(* PLC project coking-refinery, Generated TextualNotationConverter 1.0 *)
(* stored: creationDateTime 2025-07-30T12:00:00, modificationDateTime 2025-01-30T12:00:00 *)

FUNCTION_BLOCK ANALOG_IN
  VAR_INPUT
    Name : STRING;
    Description : STRING;
    Raw_Signal : REAL;
    PV_High : REAL;
    PV_Low : REAL;
    Scaling_Slope : REAL;
    Scaling_Offset : REAL;
    Alarm_Enable : BOOL;
  END_VAR
  VAR_OUTPUT
    PV : REAL;
    High_Alarm : BOOL;
    Low_Alarm : BOOL;
    General_Fault : BOOL;
  END_VAR

            
          
END_FUNCTION_BLOCK

FUNCTION_BLOCK PID_BASIC
  VAR_INPUT
    Name : STRING;
    Description : STRING;
    AUTO : BOOL;
    PV : REAL;
    SP : REAL;
    MV_MIN : REAL;
    MV_MAX : REAL;
    X0 : REAL;
    KP : REAL;
    TR : REAL;
    TD : REAL;
    PV_High : REAL;
    PV_Low : REAL;
    Deviation_Limit : REAL;
    Inhibit : BOOL;
  END_VAR
  VAR_OUTPUT
    PV_High_Alarm : BOOL;
    PV_Low_Alarm : BOOL;
    Deviation_Alarm : BOOL;
    XOUT : REAL;
  END_VAR

            
          
END_FUNCTION_BLOCK

FUNCTION_BLOCK RATIO_CONTROL
  VAR_INPUT
    Name : STRING;
    Description : STRING;
    Auto : BOOL;
    PrimaryPV : REAL;
    SecondaryPV : REAL;
    RatioSP : REAL;
    Bias : REAL;
    TrimKp : REAL;
    TrimTi : STRING;
    MV_MIN : REAL;
    MV_MAX : REAL;
    ManOut : REAL;
    Inhibit : BOOL;
  END_VAR
  VAR_OUTPUT
    SlaveSP : REAL;
    ActiveRatio : REAL;
    RatioErr : REAL;
  END_VAR

            
          
END_FUNCTION_BLOCK

FUNCTION_BLOCK VALVE_ELECTRIC
  VAR_INPUT
    Name : STRING;
    Description : STRING;
    Control_Signal : REAL;
    Manual_Mode : BOOL;
    Manual_Position : REAL;
    Open_Limit : REAL;
    Close_Limit : REAL;
    Timeout : STRING;
    Inhibit : BOOL;
  END_VAR
  VAR_OUTPUT
    Valve_Position : REAL;
    Feedback_Pos : REAL;
    Valve_Moving : BOOL;
    Position_Error : BOOL;
    Alarm : BOOL;
  END_VAR

            
          
END_FUNCTION_BLOCK

PROGRAM Section2
  VAR
    FT101_FeedFlow_PV_kgphr : REAL;
    FT102_RefluxFlow_PV_kgphr : REAL;
    FFIC103_RefluxFlow_SP_kgphr : REAL;
    FIC104_Output_Percent : REAL;
    FV104_ValvePosition_Percent : REAL;
    FV104_FeedbackPos_Percent : REAL;
    FV104_ValveMoving : BOOL;
    PIT106_ColumnPressure_bar : REAL;
    TIT104_Temperature_C : REAL;
    TIT105_Temperature_C : REAL;
    TIT107_Temperature_C : REAL;
  END_VAR
  VAR
    FT-101 : ANALOG_IN;
    FT-102 : ANALOG_IN;
    PIT-106 : ANALOG_IN;
    TIT-104 : ANALOG_IN;
    TIT-105 : ANALOG_IN;
    TIT-107 : ANALOG_IN;
    FFIC-103 : RATIO_CONTROL;
    FIC-104 : PID_BASIC;
    FV-104 : VALVE_ELECTRIC;
  END_VAR
  VAR  (* added by the conversion: wires and edge detectors of the diagram *)
    _OR1_OUT : BOOL;
  END_VAR

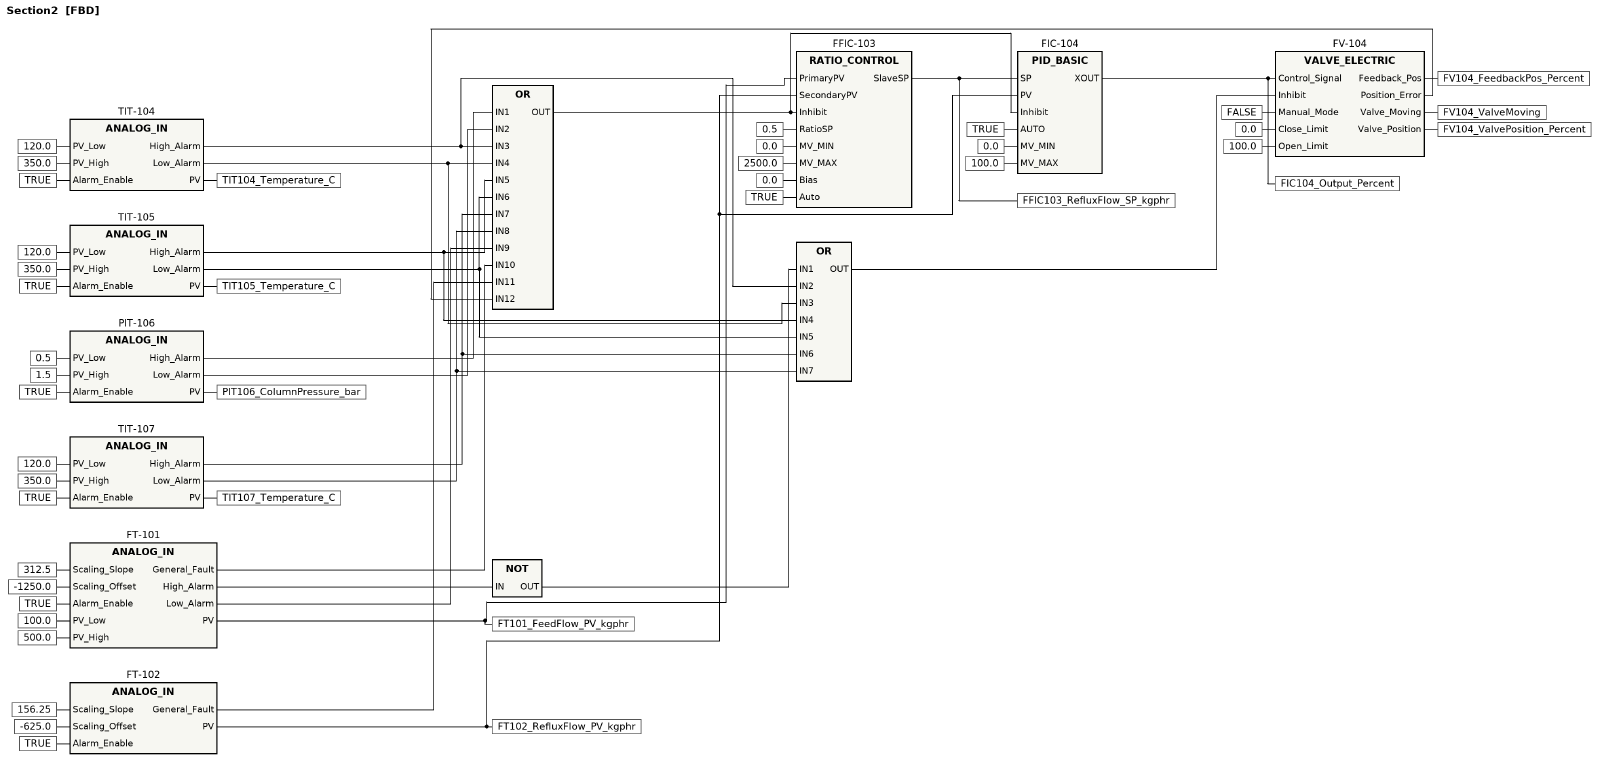
(* FBD diagram, written out as Structured Text *)
FT-101(Scaling_Slope := 312.5, Scaling_Offset := -1250.0, Alarm_Enable := TRUE, PV_Low := 100.0, PV_High := 500.0);
FT-102(Scaling_Slope := 156.25, Scaling_Offset := -625.0, Alarm_Enable := TRUE);
PIT-106(PV_Low := 0.5, PV_High := 1.5, Alarm_Enable := TRUE);
TIT-104(PV_Low := 120.0, PV_High := 350.0, Alarm_Enable := TRUE);
TIT-105(PV_Low := 120.0, PV_High := 350.0, Alarm_Enable := TRUE);
TIT-107(PV_Low := 120.0, PV_High := 350.0, Alarm_Enable := TRUE);
FIC-104(SP := FFIC-103.SlaveSP, PV := FT-102.PV, Inhibit := _OR1_OUT, AUTO := TRUE, MV_MIN := 0.0, MV_MAX := 100.0);
FV-104(Control_Signal := FIC-104.XOUT, Inhibit := NOT FT-101.High_Alarm OR TIT-104.High_Alarm OR TIT-104.Low_Alarm OR TIT-105.High_Alarm OR TIT-105.Low_Alarm OR TIT-107.High_Alarm OR TIT-107.Low_Alarm, Manual_Mode := FALSE, Close_Limit := 0.0, Open_Limit := 100.0);
_OR1_OUT := PIT-106.High_Alarm OR PIT-106.Low_Alarm OR TIT-104.High_Alarm OR TIT-104.Low_Alarm OR TIT-105.High_Alarm OR TIT-105.Low_Alarm OR TIT-107.High_Alarm OR TIT-107.Low_Alarm OR FT-101.Low_Alarm OR FT-101.General_Fault OR FT-102.General_Fault OR FV-104.Position_Error;
FFIC-103(PrimaryPV := FT-101.PV, SecondaryPV := FT-102.PV, Inhibit := _OR1_OUT, RatioSP := 0.5, MV_MIN := 0.0, MV_MAX := 2500.0, Bias := 0.0, Auto := TRUE);
FFIC103_RefluxFlow_SP_kgphr := FFIC-103.SlaveSP;
FIC104_Output_Percent := FIC-104.XOUT;
FT101_FeedFlow_PV_kgphr := FT-101.PV;
FT102_RefluxFlow_PV_kgphr := FT-102.PV;
FV104_FeedbackPos_Percent := FV-104.Feedback_Pos;
FV104_ValveMoving := FV-104.Valve_Moving;
FV104_ValvePosition_Percent := FV-104.Valve_Position;
PIT106_ColumnPressure_bar := PIT-106.PV;
TIT104_Temperature_C := TIT-104.PV;
TIT105_Temperature_C := TIT-105.PV;
TIT107_Temperature_C := TIT-107.PV;
END_PROGRAM

FUNCTION_BLOCK BOOL_IN
  VAR_INPUT
    Name : STRING;
    Description : STRING;
    Bool_In : BOOL;
    Alarm_OnTrue : BOOL;
    Alarm_OnFalse : BOOL;
    Latch_Enable : BOOL;
    Reset_Latch : BOOL;
  END_VAR
  VAR_OUTPUT
    Bool_Out : BOOL;
    Alarm_Active : BOOL;
    Latched_Status : BOOL;
  END_VAR

            
          
END_FUNCTION_BLOCK

FUNCTION_BLOCK DIGITAL_IN
  VAR_INPUT
    Name : STRING;
    Description : STRING;
    DI_Raw : BOOL;
    DebounceTime : STRING;
    EnableAlarm : BOOL;
  END_VAR
  VAR_OUTPUT
    DI_Out : BOOL;
    Fault_State : BOOL;
  END_VAR

            
          
END_FUNCTION_BLOCK

FUNCTION_BLOCK DUTY_STANDBY
  VAR_INPUT
    Name : STRING;
    Description : STRING;
    Enable : BOOL;
    StartRequest : BOOL;
    AlternateEnable : BOOL;
    ForcePumpA : BOOL;
    ForcePumpB : BOOL;
    DutyElapsed : BOOL;
    MinRunElapsed : BOOL;
    SwitchoverDelayElapsed : BOOL;
    StartTimeoutElapsed : BOOL;
    PumpA_RunFB : BOOL;
    PumpB_RunFB : BOOL;
    PumpA_Fault : BOOL;
    PumpB_Fault : BOOL;
    Reset : BOOL;
    Inhibit : BOOL;
  END_VAR
  VAR_OUTPUT
    CmdPumpA : BOOL;
    CmdPumpB : BOOL;
    ActiveIsA : BOOL;
    SwitchedDueToDuty : BOOL;
    SwitchedDueToFailure : BOOL;
    Alarm_FailedStart_A : BOOL;
    Alarm_FailedStart_B : BOOL;
    Alarm_NoAvailablePump : BOOL;
  END_VAR

            
          
END_FUNCTION_BLOCK

FUNCTION_BLOCK MOTOR_2SPD
  VAR_INPUT
    Name : STRING;
    Description : STRING;
    Start_Cmd : BOOL;
    Stop_Cmd : BOOL;
    Speed_High_Cmd : BOOL;
    Speed_Low_Cmd : BOOL;
    Inhibit : BOOL;
  END_VAR
  VAR_OUTPUT
    Motor_Start_Out : BOOL;
    FB_Running : BOOL;
    FB_Trip : BOOL;
    FB_HighSpeed : BOOL;
    FB_LowSpeed : BOOL;
    Alarm_Speed_Error : BOOL;
  END_VAR

            
          
END_FUNCTION_BLOCK

FUNCTION_BLOCK MOTOR_ON_OFF
  VAR_INPUT
    Name : STRING;
    Description : STRING;
    Start_Cmd : BOOL;
    Stop_Cmd : BOOL;
    Start_Delay : STRING;
    MinRunTime : STRING;
    Inhibit : BOOL;
  END_VAR
  VAR_OUTPUT
    Motor_Start_Out : BOOL;
    FB_Running : BOOL;
    FB_Trip : BOOL;
    Alarm_Start_Fail : BOOL;
    Alarm_Stop_Fail : BOOL;
  END_VAR

            
          
END_FUNCTION_BLOCK

FUNCTION_BLOCK MOTOR_VSD
  VAR_INPUT
    Name : STRING;
    Description : STRING;
    Start_Cmd : BOOL;
    Stop_Cmd : BOOL;
    Speed_SP : REAL;
    Accel_Ramp : STRING;
    Decel_Ramp : STRING;
    Inhibit : BOOL;
  END_VAR
  VAR_OUTPUT
    Speed_Out : REAL;
    FB_Running : BOOL;
    FB_Fault : BOOL;
    FB_Ready : BOOL;
    FB_ActualSpeed : REAL;
    Alarm_Speed_Deviation : BOOL;
    Alarm_Comm_Fail : BOOL;
  END_VAR

            
          
END_FUNCTION_BLOCK

FUNCTION_BLOCK SPLIT_RANGE
  VAR_INPUT
    Name : STRING;
    Description : STRING;
    IN : REAL;
    Split_Point : REAL;
    Output1_Start : REAL;
    Output1_End : REAL;
    Output2_Start : REAL;
    Output2_End : REAL;
  END_VAR
  VAR_OUTPUT
    OUT1 : REAL;
    OUT2 : REAL;
  END_VAR

            
          
END_FUNCTION_BLOCK

FUNCTION_BLOCK VALVE_ON_OFF
  VAR_INPUT
    Name : STRING;
    Description : STRING;
    Open_Cmd : BOOL;
    Close_Cmd : BOOL;
    Timeout : STRING;
    Inhibit : BOOL;
  END_VAR
  VAR_OUTPUT
    FB_Opened : BOOL;
    FB_Closed : BOOL;
    Valve_Open_Out : BOOL;
    Valve_Close_Out : BOOL;
    Alarm_Position_Error : BOOL;
    Alarm_General : BOOL;
  END_VAR

            
          
END_FUNCTION_BLOCK

FUNCTION_BLOCK VOTING_ANALOG
  VAR_INPUT
    Name : STRING;
    Description : STRING;
    Input1 : REAL;
    Input2 : REAL;
    Input3 : REAL;
    Deviation_Limit : REAL;
    Voting_Scheme : STRING;
    EnableAlarm : BOOL;
    Inhibit : BOOL;
  END_VAR
  VAR_OUTPUT
    Voted_Output : REAL;
    Sensor1_Fault : BOOL;
    Sensor2_Fault : BOOL;
    Sensor3_Fault : BOOL;
    Alarm_Voting_Error : BOOL;
    Healthy_Sensors_Count : INT;
  END_VAR

            
          
END_FUNCTION_BLOCK

PROGRAM Section3
  VAR
    PIT_103_PV_mmHg : REAL;
    PIC_102_MV_Percent : REAL;
  END_VAR
  VAR
    PIT-103 : ANALOG_IN;
    PIC-102 : PID_BASIC;
    PV-101 : VALVE_ELECTRIC;
    VDU_START_OK : BOOL_IN;
    MAINT_BYPASS_OK : BOOL_IN;
  END_VAR
  VAR  (* added by the conversion: wires and edge detectors of the diagram *)
    _OR56_OUT : BOOL;
  END_VAR

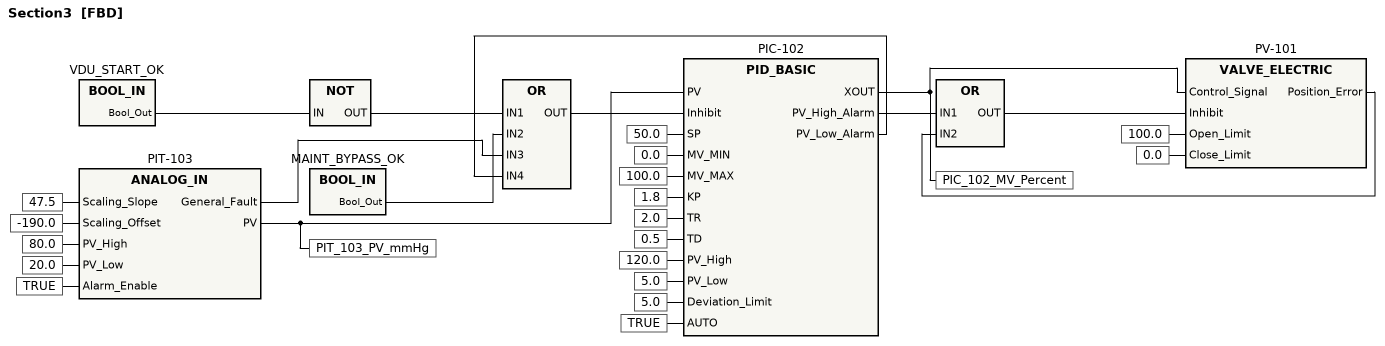
(* FBD diagram, written out as Structured Text *)
PIT-103(Scaling_Slope := 47.5, Scaling_Offset := -190.0, PV_High := 80.0, PV_Low := 20.0, Alarm_Enable := TRUE);
VDU_START_OK();
MAINT_BYPASS_OK();
PIC-102(PV := PIT-103.PV, Inhibit := NOT VDU_START_OK.Bool_Out OR MAINT_BYPASS_OK.Bool_Out OR PIT-103.General_Fault OR PIC-102.PV_Low_Alarm, SP := 50.0, MV_MIN := 0.0, MV_MAX := 100.0, KP := 1.8, TR := 2.0, TD := 0.5, PV_High := 120.0, PV_Low := 5.0, Deviation_Limit := 5.0, AUTO := TRUE);
PIC_102_MV_Percent := PIC-102.XOUT;
PIT_103_PV_mmHg := PIT-103.PV;
PV-101(Control_Signal := PIC-102.XOUT, Inhibit := _OR56_OUT, Open_Limit := 100.0, Close_Limit := 0.0);
_OR56_OUT := PIC-102.PV_High_Alarm OR PV-101.Position_Error;
END_PROGRAM

PROGRAM Section4
  VAR
    PC301_SP_Operator : REAL;
    PT_301_RegeneratorPressure_PV : REAL;
    PT_302_BlowerDischargePressure_PV : REAL;
    PT_303_FractionatorOverheadPressure_PV : REAL;
    TT_301_RegeneratorTemperature_PV : REAL;
    PTF_301_FilteredPressure_PV : REAL;
    PC_301_Output_to_PV_105_Percent : REAL;
    PV_105_Valve_Position_Command_Percent : REAL;
    PV_105_Valve_Position_Feedback_Percent : REAL;
    P_301A_Running_Status : BOOL;
    XV_108_Closed_Status : BOOL;
  END_VAR
  VAR
    PT-301 : ANALOG_IN;
    PT-302 : ANALOG_IN;
    PT-303 : ANALOG_IN;
    PTF-301 : ANALOG_IN;
    TT-301 : ANALOG_IN;
    PC-301 : PID_BASIC;
    PV-105 : VALVE_ELECTRIC;
    PV-106 : VALVE_ON_OFF;
    XV-108 : VALVE_ON_OFF;
    P-301A : MOTOR_ON_OFF;
    SteadyState_TON : TON;
  END_VAR
  VAR  (* added by the conversion: wires and edge detectors of the diagram *)
    _SEL83_OUT : ANY;
    _SUB84_OUT : REAL;
    _OR87_OUT : BOOL;
    _LIMIT82_OUT : REAL;
    _GT98_OUT : BOOL;
  END_VAR

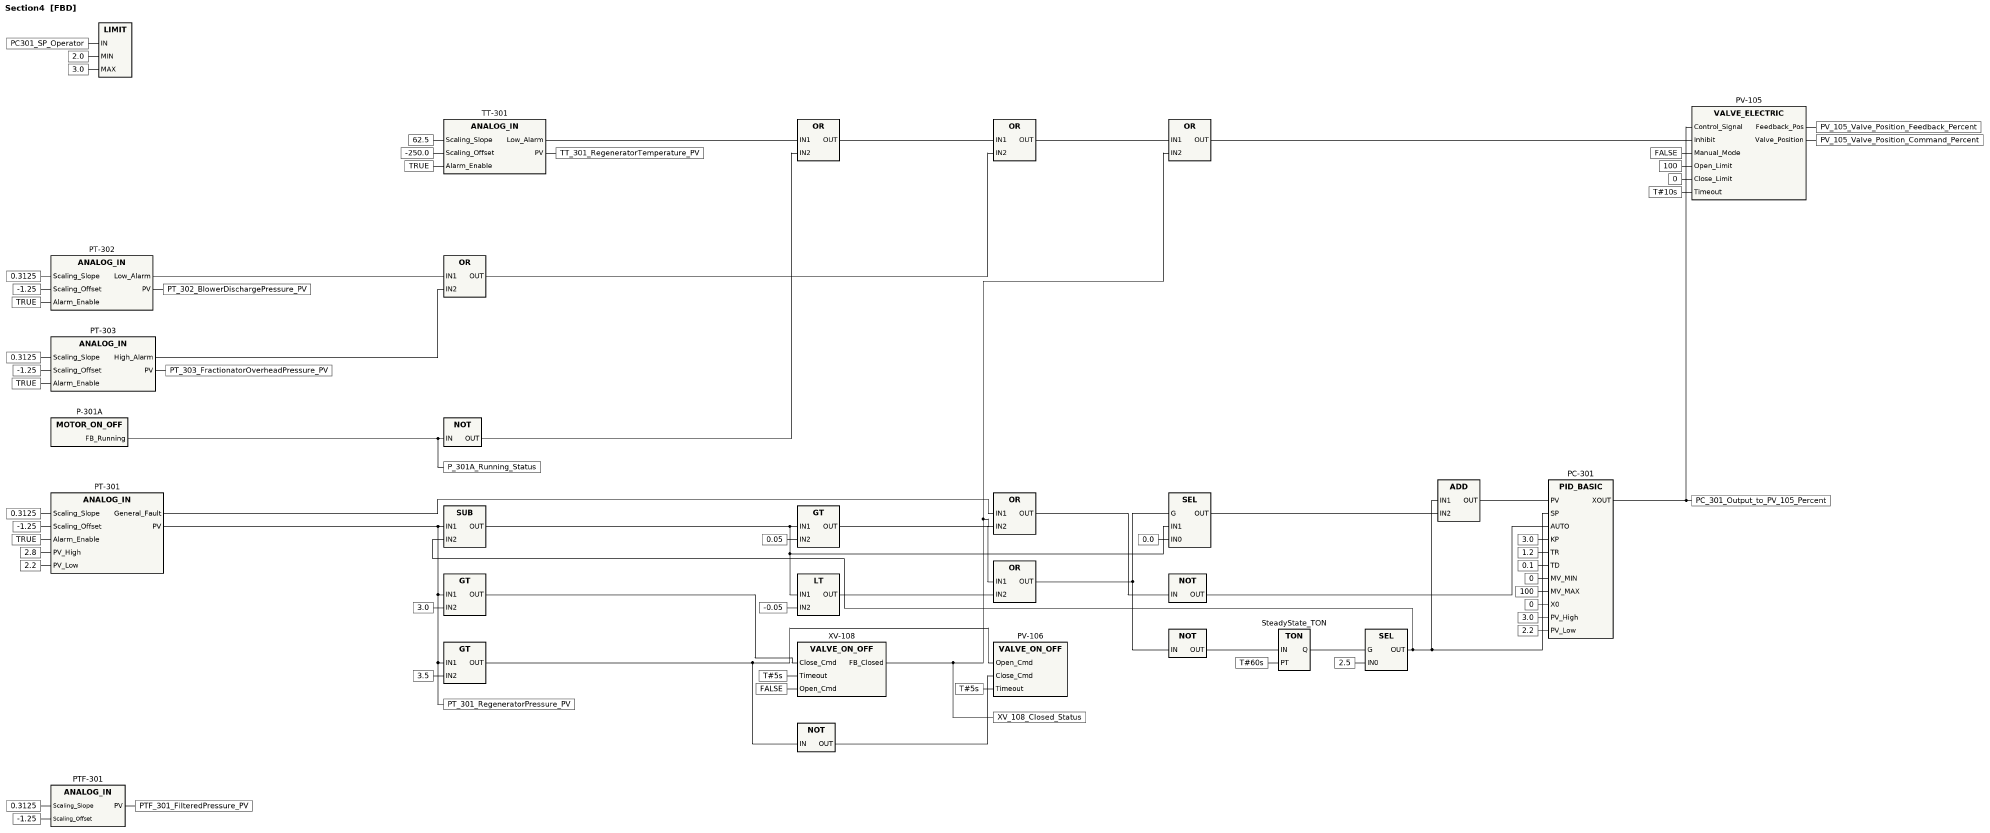
(* FBD diagram, written out as Structured Text *)
PT-301(Scaling_Slope := 0.3125, Scaling_Offset := -1.25, Alarm_Enable := TRUE, PV_High := 2.8, PV_Low := 2.2);
_SUB84_OUT := PT-301.PV - _SEL83_OUT;
_OR87_OUT := _SUB84_OUT > 0.05 OR _SUB84_OUT < (-0.05);
SteadyState_TON(IN := NOT _OR87_OUT, PT := T#60s);
_SEL83_OUT := SEL(SteadyState_TON.Q, 2.5);
XV-108(Close_Cmd := PT-301.PV > 3.0, Timeout := T#5s, Open_Cmd := FALSE);
PC-301(PV := _SEL83_OUT + SEL(_OR87_OUT, _SUB84_OUT, 0.0), SP := _SEL83_OUT, AUTO := NOT (PT-301.General_Fault OR XV-108.FB_Closed), KP := 3.0, TR := 1.2, TD := 0.1, MV_MIN := 0, MV_MAX := 100, X0 := 0, PV_High := 3.0, PV_Low := 2.2);
PC_301_Output_to_PV_105_Percent := PC-301.XOUT;
PTF-301(Scaling_Slope := 0.3125, Scaling_Offset := -1.25);
PTF_301_FilteredPressure_PV := PTF-301.PV;
PT_301_RegeneratorPressure_PV := PT-301.PV;
PT-302(Scaling_Slope := 0.3125, Scaling_Offset := -1.25, Alarm_Enable := TRUE);
PT_302_BlowerDischargePressure_PV := PT-302.PV;
PT-303(Scaling_Slope := 0.3125, Scaling_Offset := -1.25, Alarm_Enable := TRUE);
PT_303_FractionatorOverheadPressure_PV := PT-303.PV;
TT-301(Scaling_Slope := 62.5, Scaling_Offset := -250.0, Alarm_Enable := TRUE);
P-301A();
PV-105(Control_Signal := PC-301.XOUT, Inhibit := TT-301.Low_Alarm OR NOT P-301A.FB_Running OR PT-302.Low_Alarm OR PT-303.High_Alarm OR XV-108.FB_Closed, Manual_Mode := FALSE, Open_Limit := 100, Close_Limit := 0, Timeout := T#10s);
PV_105_Valve_Position_Command_Percent := PV-105.Valve_Position;
PV_105_Valve_Position_Feedback_Percent := PV-105.Feedback_Pos;
P_301A_Running_Status := P-301A.FB_Running;
TT_301_RegeneratorTemperature_PV := TT-301.PV;
XV_108_Closed_Status := XV-108.FB_Closed;
_LIMIT82_OUT := LIMIT(PC301_SP_Operator, 2.0, 3.0);
_GT98_OUT := PT-301.PV > 3.5;
PV-106(Open_Cmd := _GT98_OUT, Close_Cmd := NOT _GT98_OUT, Timeout := T#5s);
END_PROGRAM

PROGRAM Section5
  VAR
    TIT101_FurnaceOutletTemp_PV_C : REAL;
    TC401_FV401_FuelGas_MV_Pct : REAL;
    PT402_FurnaceDraft_PV_kPa : REAL;
    PT403_DischargePressure_PV_bar : REAL;
    PC401_FuelGasPressure_PV_bar : REAL;
    TIT101_HighTempAlarm_3s : BOOL;
    TIT101_LowTempAlarm_3s : BOOL;
  END_VAR
  VAR
    TIT-101 : ANALOG_IN;
    TC-401 : PID_BASIC;
    FV-401 : VALVE_ELECTRIC;
    PT-402 : ANALOG_IN;
    PT-403 : ANALOG_IN;
    PC-401 : PID_BASIC;
    FT-401A : DIGITAL_IN;
    FT-401B : DIGITAL_IN;
    FuelGasInterlockDelay_TON : TON;
    TIT101_HighAlarmDelay_TON : TON;
    TIT101_LowAlarmDelay_TON : TON;
  END_VAR
  VAR  (* added by the conversion: wires and edge detectors of the diagram *)
    _OR166_OUT : BOOL;
  END_VAR

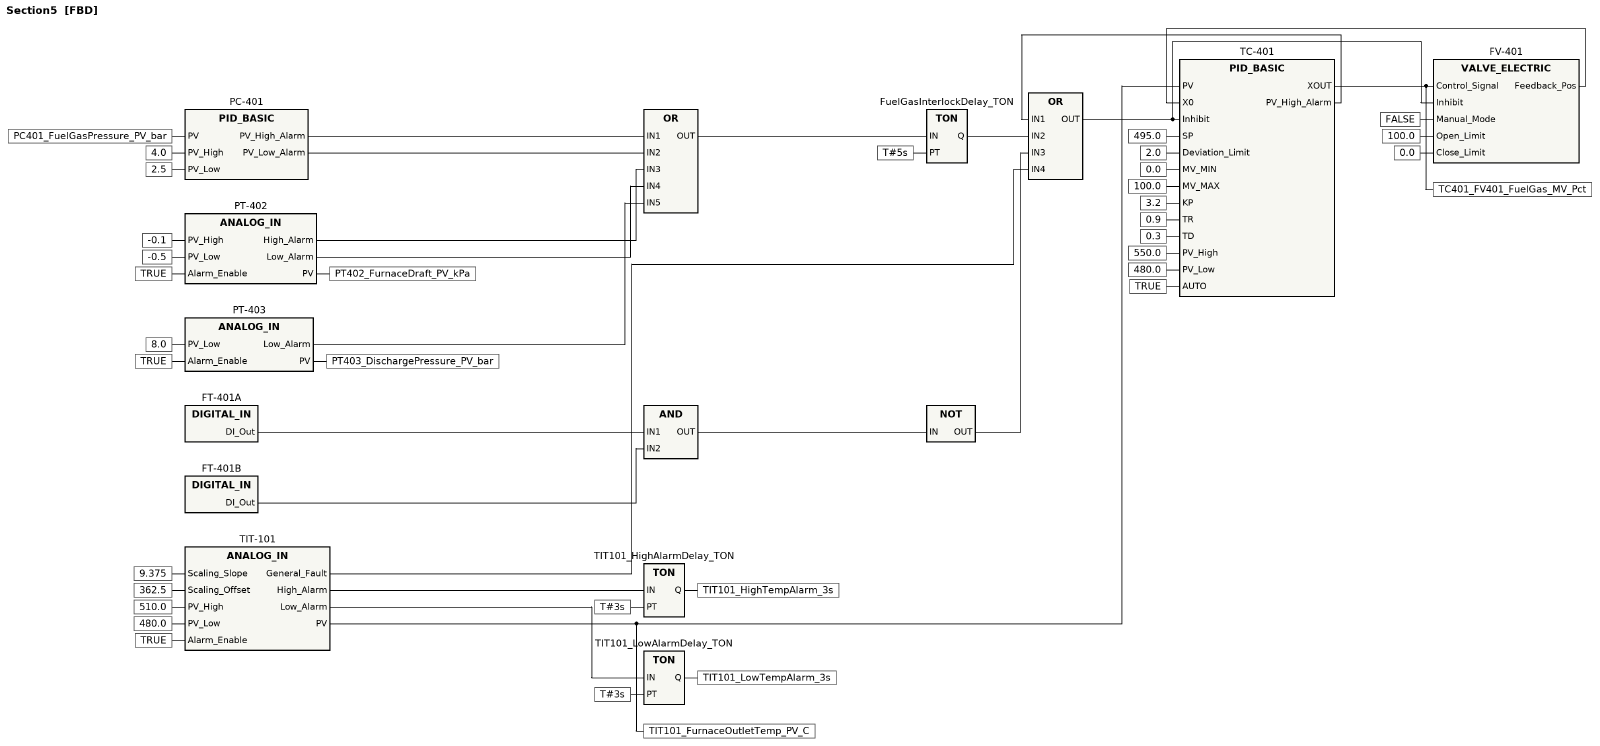
(* FBD diagram, written out as Structured Text *)
PT-402(PV_High := -0.1, PV_Low := -0.5, Alarm_Enable := TRUE);
PT402_FurnaceDraft_PV_kPa := PT-402.PV;
PT-403(PV_Low := 8.0, Alarm_Enable := TRUE);
PT403_DischargePressure_PV_bar := PT-403.PV;
TIT-101(Scaling_Slope := 9.375, Scaling_Offset := 362.5, PV_High := 510.0, PV_Low := 480.0, Alarm_Enable := TRUE);
PC-401(PV := PC401_FuelGasPressure_PV_bar, PV_High := 4.0, PV_Low := 2.5);
FuelGasInterlockDelay_TON(IN := PC-401.PV_High_Alarm OR PC-401.PV_Low_Alarm OR PT-402.High_Alarm OR PT-402.Low_Alarm OR PT-403.Low_Alarm, PT := T#5s);
FT-401A();
FT-401B();
_OR166_OUT := TC-401.PV_High_Alarm OR FuelGasInterlockDelay_TON.Q OR NOT (FT-401A.DI_Out AND FT-401B.DI_Out) OR TIT-101.General_Fault;
FV-401(Control_Signal := TC-401.XOUT, Inhibit := _OR166_OUT, Manual_Mode := FALSE, Open_Limit := 100.0, Close_Limit := 0.0);
TC-401(PV := TIT-101.PV, X0 := FV-401.Feedback_Pos, Inhibit := _OR166_OUT, SP := 495.0, Deviation_Limit := 2.0, MV_MIN := 0.0, MV_MAX := 100.0, KP := 3.2, TR := 0.9, TD := 0.3, PV_High := 550.0, PV_Low := 480.0, AUTO := TRUE);
TC401_FV401_FuelGas_MV_Pct := TC-401.XOUT;
TIT101_FurnaceOutletTemp_PV_C := TIT-101.PV;
TIT101_HighAlarmDelay_TON(IN := TIT-101.High_Alarm, PT := T#3s);
TIT101_HighTempAlarm_3s := TIT101_HighAlarmDelay_TON.Q;
TIT101_LowAlarmDelay_TON(IN := TIT-101.Low_Alarm, PT := T#3s);
TIT101_LowTempAlarm_3s := TIT101_LowAlarmDelay_TON.Q;
END_PROGRAM

PROGRAM Section6
  VAR
    FT103_H2Flow_PV : REAL;
    FC103_MV_Percent : REAL;
    TT101_Temp_PV : REAL;
    TC501_MV_Percent : REAL;
    PT501_Pressure_PV : REAL;
    PT502_InletPressure_PV : REAL;
    FC103_SP_Operator : REAL;
    FC103_SP_Clamped : REAL;
    FC103_SP_Reduced : REAL;
  END_VAR
  VAR
    FT-103 : ANALOG_IN;
    FC-103 : PID_BASIC;
    FV-103 : VALVE_ELECTRIC;
    TT-101 : ANALOG_IN;
    TC-501 : PID_BASIC;
    TV-501 : VALVE_ELECTRIC;
    PT-501 : ANALOG_IN;
    PC-501 : PID_BASIC;
    PT-502 : ANALOG_IN;
    ESD-501 : DIGITAL_IN;
  END_VAR
  VAR  (* added by the conversion: wires and edge detectors of the diagram *)
    _OR213_OUT : BOOL;
    _OR219_OUT : BOOL;
    _MIN229_OUT : REAL;
    _NOT221_OUT : BOOL;
  END_VAR

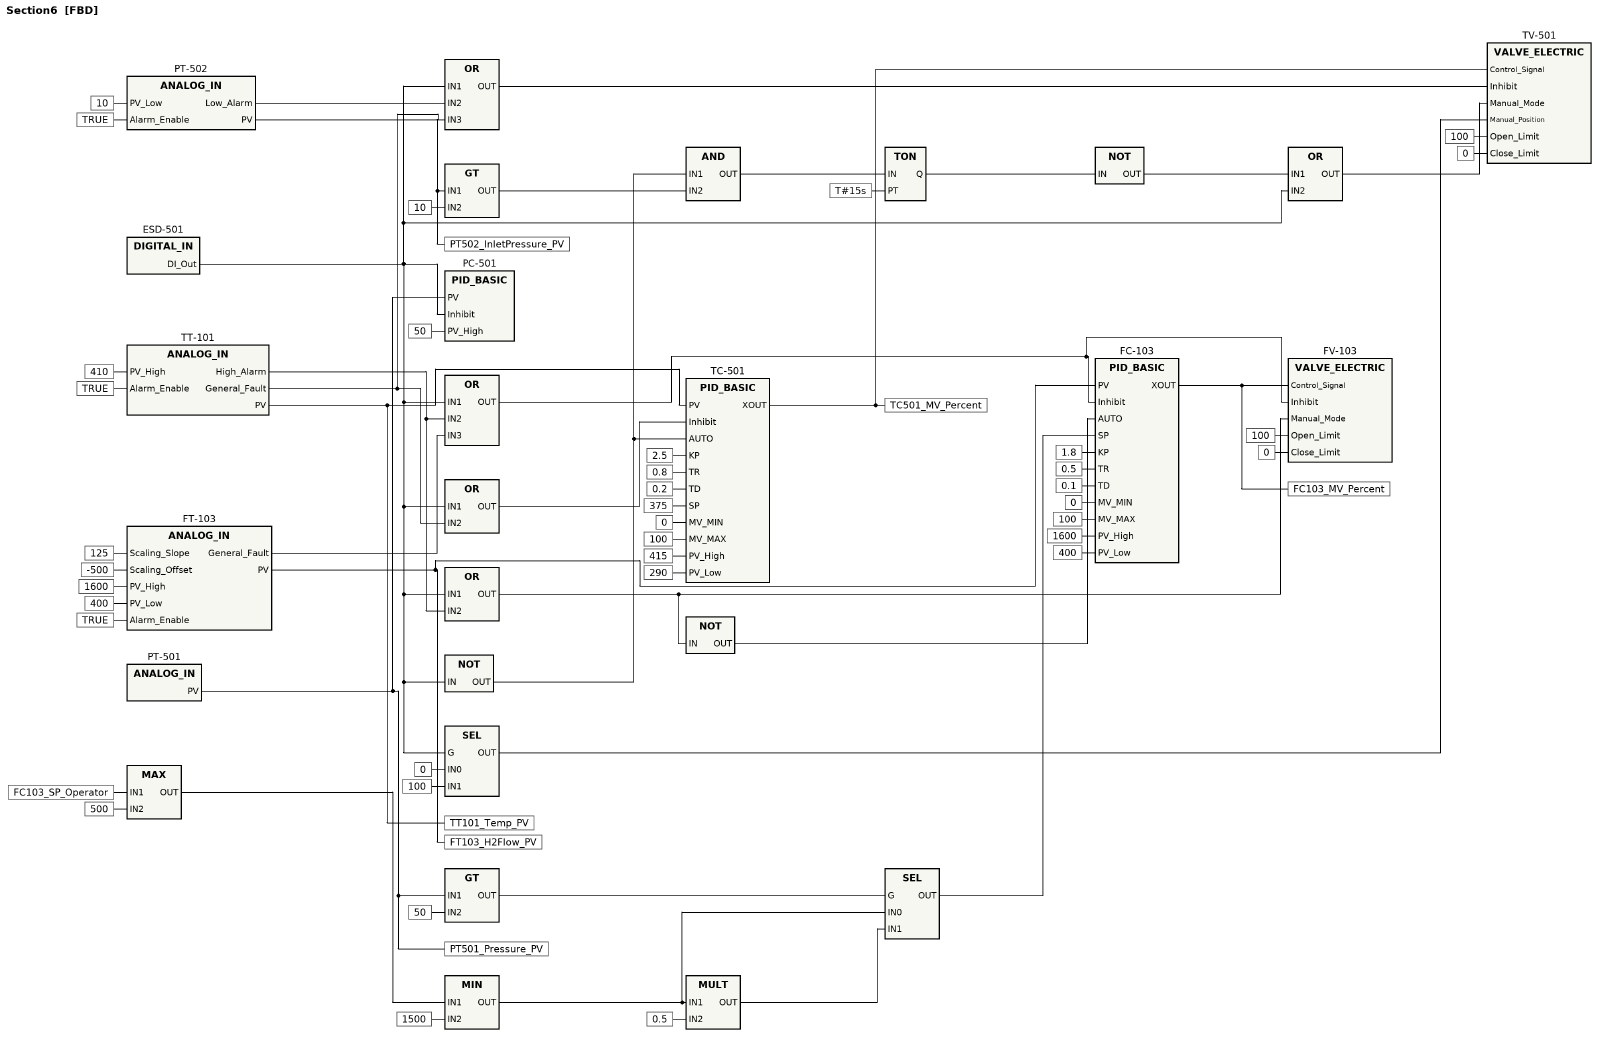
(* FBD diagram, written out as Structured Text *)
FT-103(Scaling_Slope := 125, Scaling_Offset := -500, PV_High := 1600, PV_Low := 400, Alarm_Enable := TRUE);
ESD-501();
TT-101(PV_High := 410, Alarm_Enable := TRUE);
_OR213_OUT := ESD-501.DI_Out OR TT-101.High_Alarm OR FT-103.General_Fault;
_OR219_OUT := ESD-501.DI_Out OR TT-101.High_Alarm;
PT-501();
_MIN229_OUT := MIN(MAX(FC103_SP_Operator, 500), 1500);
FC-103(PV := FT-103.PV, Inhibit := _OR213_OUT, AUTO := NOT _OR219_OUT, SP := SEL(PT-501.PV > 50, _MIN229_OUT, MULT(_MIN229_OUT, 0.5)), KP := 1.8, TR := 0.5, TD := 0.1, MV_MIN := 0, MV_MAX := 100, PV_High := 1600, PV_Low := 400);
FC103_MV_Percent := FC-103.XOUT;
FT103_H2Flow_PV := FT-103.PV;
PT501_Pressure_PV := PT-501.PV;
PT-502(PV_Low := 10, Alarm_Enable := TRUE);
PT502_InletPressure_PV := PT-502.PV;
_NOT221_OUT := NOT ESD-501.DI_Out;
TC-501(PV := TT-101.PV, Inhibit := ESD-501.DI_Out OR TT-101.General_Fault, AUTO := _NOT221_OUT, KP := 2.5, TR := 0.8, TD := 0.2, SP := 375, MV_MIN := 0, MV_MAX := 100, PV_High := 415, PV_Low := 290);
TC501_MV_Percent := TC-501.XOUT;
TT101_Temp_PV := TT-101.PV;
FV-103(Control_Signal := FC-103.XOUT, Inhibit := _OR213_OUT, Manual_Mode := _OR219_OUT, Open_Limit := 100, Close_Limit := 0);
TV-501(Control_Signal := TC-501.XOUT, Inhibit := ESD-501.DI_Out OR PT-502.Low_Alarm OR TT-101.General_Fault, Manual_Mode := NOT TON(_NOT221_OUT AND PT-502.PV > 10, T#15s) OR ESD-501.DI_Out, Manual_Position := SEL(ESD-501.DI_Out, 0, 100), Open_Limit := 100, Close_Limit := 0);
PC-501(PV := PT-501.PV, Inhibit := ESD-501.DI_Out, PV_High := 50);
END_PROGRAM

PROGRAM Section7
  VAR
    FT601_Raw_mA : REAL;
    LT601_Raw_mA : REAL;
    TT104_Raw_mA : REAL;
    FT601_FlowRate_m3h_PV : REAL;
    LT601_SiloLevel_Pct_PV : REAL;
    TT104_Temperature_C_PV : REAL;
    FIC601_MV_Pct : REAL;
    P601A_SpeedCmd_Pct : REAL;
    P601B_SpeedCmd_Pct : REAL;
    SP_Operator_m3h : REAL;
    FA601_LowFlow_Alarm : BOOL;
    LAH601_HighLevel_Alarm : BOOL;
    TAH104_HighTemp_Alarm : BOOL;
    Start_Pumps_Cmd : BOOL;
    Stop_Pumps_Cmd : BOOL;
    MCC601_Status_In : BOOL;
    MCC602_Status_In : BOOL;
    Crusher_RunPermissive : BOOL;
    Permissive_All_OK : BOOL;
    FT601_Signal_OK : BOOL;
  END_VAR
  VAR
    FT-601 : ANALOG_IN;
    LT-601 : ANALOG_IN;
    TT-104 : ANALOG_IN;
    FIC-601 : PID_BASIC;
    P-601A : MOTOR_VSD;
    P-601B : MOTOR_VSD;
    MCC-601 : BOOL_IN;
    MCC-602 : BOOL_IN;
    StartDelay_TON : TON;
    LowFlowDelay_TON : TON;
  END_VAR
  VAR  (* added by the conversion: wires and edge detectors of the diagram *)
    _NOT288_OUT : BOOL;
    _OR284_OUT : BOOL;
    _OR292_OUT : BOOL;
  END_VAR

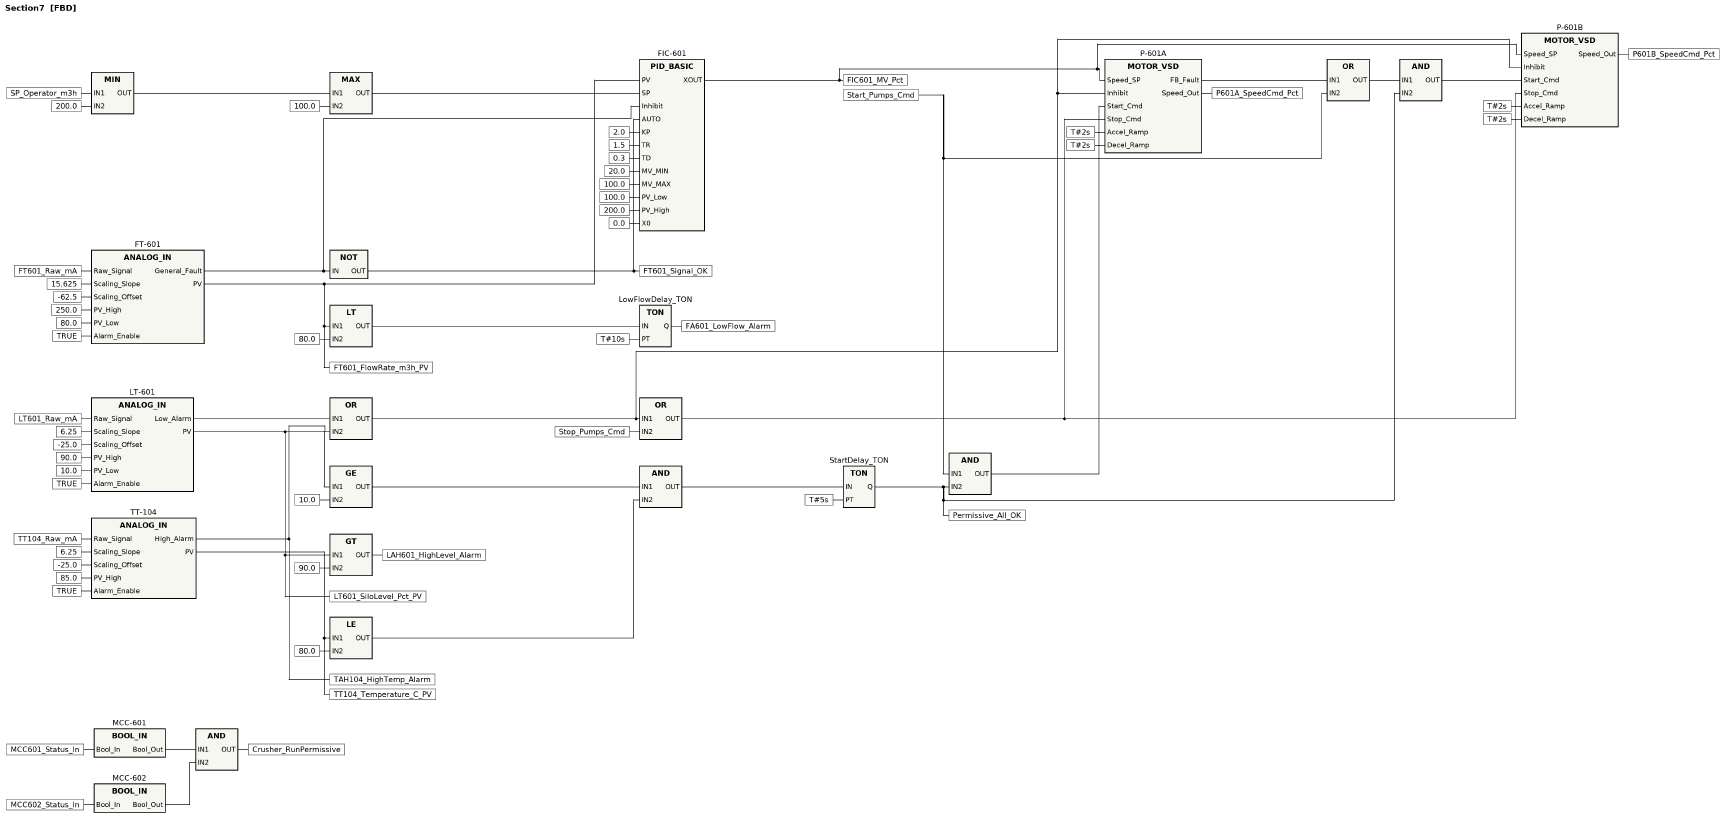
(* FBD diagram, written out as Structured Text *)
MCC-601(Bool_In := MCC601_Status_In);
MCC-602(Bool_In := MCC602_Status_In);
Crusher_RunPermissive := MCC-601.Bool_Out AND MCC-602.Bool_Out;
FT-601(Raw_Signal := FT601_Raw_mA, Scaling_Slope := 15.625, Scaling_Offset := -62.5, PV_High := 250.0, PV_Low := 80.0, Alarm_Enable := TRUE);
LowFlowDelay_TON(IN := FT-601.PV < 80.0, PT := T#10s);
FA601_LowFlow_Alarm := LowFlowDelay_TON.Q;
_NOT288_OUT := NOT FT-601.General_Fault;
FIC-601(PV := FT-601.PV, SP := MAX(MIN(SP_Operator_m3h, 200.0), 100.0), Inhibit := FT-601.General_Fault, AUTO := _NOT288_OUT, KP := 2.0, TR := 1.5, TD := 0.3, MV_MIN := 20.0, MV_MAX := 100.0, PV_Low := 100.0, PV_High := 200.0, X0 := 0.0);
FIC601_MV_Pct := FIC-601.XOUT;
FT601_FlowRate_m3h_PV := FT-601.PV;
FT601_Signal_OK := _NOT288_OUT;
LT-601(Raw_Signal := LT601_Raw_mA, Scaling_Slope := 6.25, Scaling_Offset := -25.0, PV_High := 90.0, PV_Low := 10.0, Alarm_Enable := TRUE);
LAH601_HighLevel_Alarm := LT-601.PV > 90.0;
LT601_SiloLevel_Pct_PV := LT-601.PV;
TT-104(Raw_Signal := TT104_Raw_mA, Scaling_Slope := 6.25, Scaling_Offset := -25.0, PV_High := 85.0, Alarm_Enable := TRUE);
_OR284_OUT := LT-601.Low_Alarm OR TT-104.High_Alarm;
StartDelay_TON(IN := LT-601.PV >= 10.0 AND TT-104.PV <= 80.0, PT := T#5s);
_OR292_OUT := _OR284_OUT OR Stop_Pumps_Cmd;
P-601A(Speed_SP := FIC-601.XOUT, Inhibit := _OR284_OUT, Start_Cmd := Start_Pumps_Cmd AND StartDelay_TON.Q, Stop_Cmd := _OR292_OUT, Accel_Ramp := T#2s, Decel_Ramp := T#2s);
P601A_SpeedCmd_Pct := P-601A.Speed_Out;
P-601B(Speed_SP := FIC-601.XOUT, Inhibit := _OR284_OUT, Start_Cmd := (P-601A.FB_Fault OR Start_Pumps_Cmd) AND StartDelay_TON.Q, Stop_Cmd := _OR292_OUT, Accel_Ramp := T#2s, Decel_Ramp := T#2s);
P601B_SpeedCmd_Pct := P-601B.Speed_Out;
Permissive_All_OK := StartDelay_TON.Q;
TAH104_HighTemp_Alarm := TT-104.High_Alarm;
TT104_Temperature_C_PV := TT-104.PV;
END_PROGRAM

PROGRAM Section8
  VAR
    FT702_AirFlow_SP : REAL;
  END_VAR
  VAR
    FT-701 : ANALOG_IN;
    FT-702 : ANALOG_IN;
    PT-701 : ANALOG_IN;
    FD-701 : BOOL_IN;
    FFIC-701 : RATIO_CONTROL;
    FIC-702 : PID_BASIC;
    LIC-101 : PID_BASIC;
    FV-701 : VALVE_ELECTRIC;
    FV-702 : VALVE_ELECTRIC;
  END_VAR
  VAR  (* added by the conversion: wires and edge detectors of the diagram *)
    _OR365_OUT : BOOL;
  END_VAR

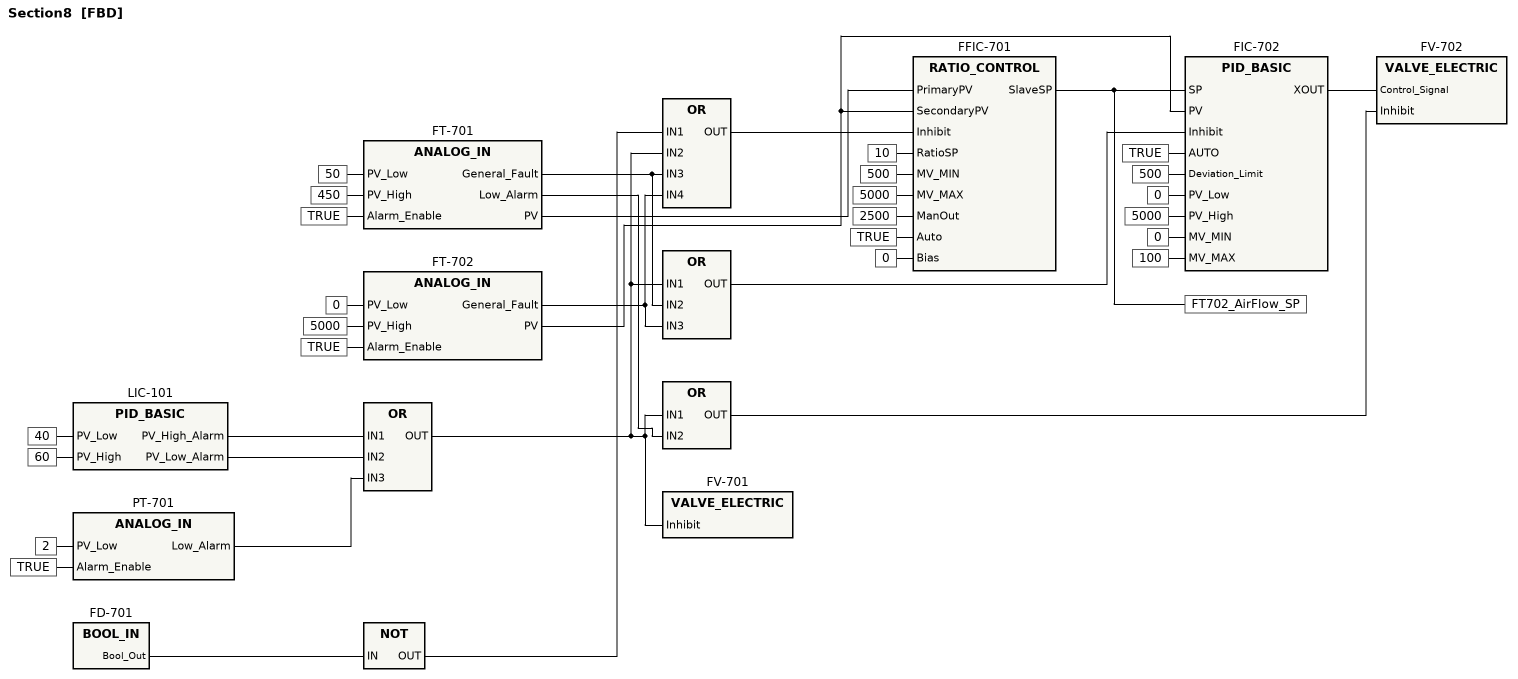
(* FBD diagram, written out as Structured Text *)
FT-701(PV_Low := 50, PV_High := 450, Alarm_Enable := TRUE);
FT-702(PV_Low := 0, PV_High := 5000, Alarm_Enable := TRUE);
FD-701();
LIC-101(PV_Low := 40, PV_High := 60);
PT-701(PV_Low := 2, Alarm_Enable := TRUE);
_OR365_OUT := LIC-101.PV_High_Alarm OR LIC-101.PV_Low_Alarm OR PT-701.Low_Alarm;
FFIC-701(PrimaryPV := FT-701.PV, SecondaryPV := FT-702.PV, Inhibit := NOT FD-701.Bool_Out OR _OR365_OUT OR FT-701.General_Fault OR FT-702.General_Fault, RatioSP := 10, MV_MIN := 500, MV_MAX := 5000, ManOut := 2500, Auto := TRUE, Bias := 0);
FT702_AirFlow_SP := FFIC-701.SlaveSP;
FIC-702(SP := FFIC-701.SlaveSP, PV := FT-702.PV, Inhibit := _OR365_OUT OR FT-701.General_Fault OR FT-702.General_Fault, AUTO := TRUE, Deviation_Limit := 500, PV_Low := 0, PV_High := 5000, MV_MIN := 0, MV_MAX := 100);
FV-701(Inhibit := _OR365_OUT);
FV-702(Control_Signal := FIC-702.XOUT, Inhibit := _OR365_OUT OR FT-701.Low_Alarm);
END_PROGRAM

PROGRAM Section9
  VAR
    PT106_PV_Pct : REAL;
    PIC101_MV_Pct : REAL;
    FV102_Feedback_Pos_Pct : REAL;
  END_VAR
  VAR
    PT-106 : ANALOG_IN;
    PIC-101 : PID_BASIC;
    FV-102 : VALVE_ELECTRIC;
    LC-801_LEVEL_OK : BOOL_IN;
    FLARE_IGNITION_OK : BOOL_IN;
    PT-106_VALID : BOOL_IN;
  END_VAR

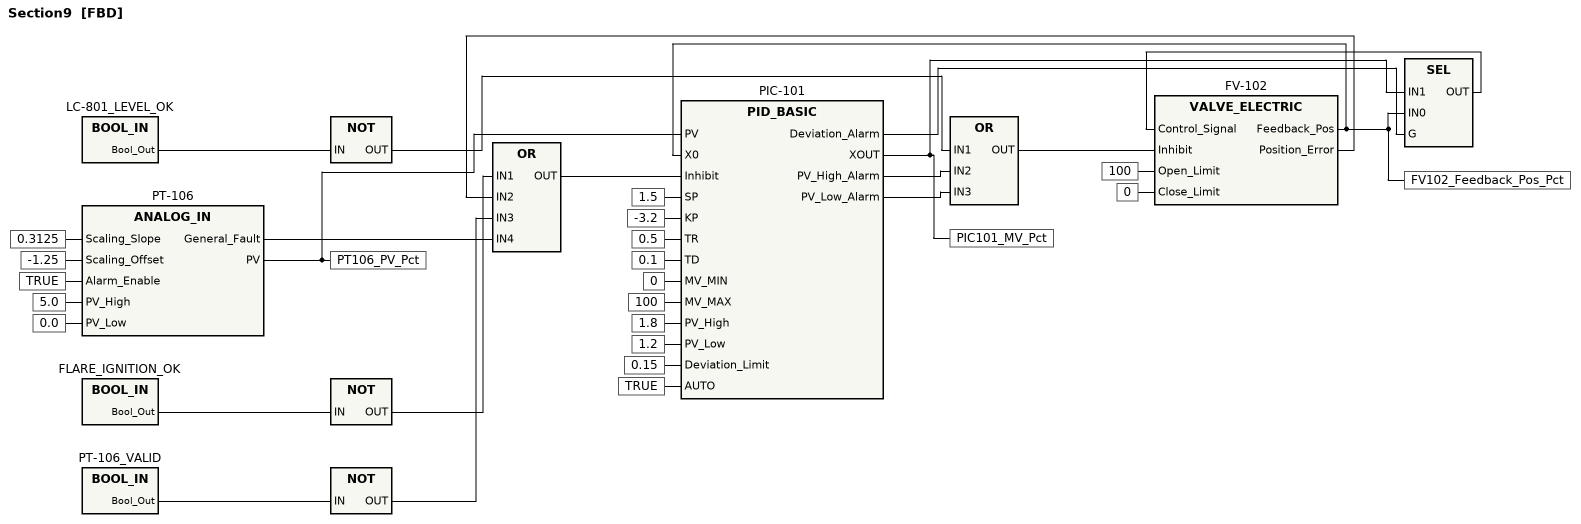
(* FBD diagram, written out as Structured Text *)
PT-106(Scaling_Slope := 0.3125, Scaling_Offset := -1.25, Alarm_Enable := TRUE, PV_High := 5.0, PV_Low := 0.0);
FLARE_IGNITION_OK();
PT-106_VALID();
PIC-101(PV := PT-106.PV, X0 := FV-102.Feedback_Pos, Inhibit := NOT FLARE_IGNITION_OK.Bool_Out OR FV-102.Position_Error OR NOT PT-106_VALID.Bool_Out OR PT-106.General_Fault, SP := 1.5, KP := -3.2, TR := 0.5, TD := 0.1, MV_MIN := 0, MV_MAX := 100, PV_High := 1.8, PV_Low := 1.2, Deviation_Limit := 0.15, AUTO := TRUE);
LC-801_LEVEL_OK();
FV-102(Control_Signal := SEL(PIC-101.XOUT, FV-102.Feedback_Pos, PIC-101.Deviation_Alarm), Inhibit := NOT LC-801_LEVEL_OK.Bool_Out OR PIC-101.PV_High_Alarm OR PIC-101.PV_Low_Alarm, Open_Limit := 100, Close_Limit := 0);
FV102_Feedback_Pos_Pct := FV-102.Feedback_Pos;
PIC101_MV_Pct := PIC-101.XOUT;
PT106_PV_Pct := PT-106.PV;
END_PROGRAM

CONFIGURATION Config0
  RESOURCE Res0 ON PLC
    TASK task0(INTERVAL := T#20ms, PRIORITY := 0);
    PROGRAM instance0 WITH task0 : Section2;
    PROGRAM instance_1 WITH task0 : Section3;
    PROGRAM instance_2 WITH task0 : Section4;
    PROGRAM instance_3 WITH task0 : Section5;
    PROGRAM instance_4 WITH task0 : Section6;
    PROGRAM instance_5 WITH task0 : Section7;
    PROGRAM instance_6 WITH task0 : Section8;
    PROGRAM instance_7 WITH task0 : Section9;
  END_RESOURCE
END_CONFIGURATION
